(* IEC 61131-3 sources: Simulated-machine/integrations/openplc/thermal-plant-v4/pous/programs (part 2) *)

  (* Rising-edge plant trip matrix, matching examples/external_plc.py. *)
  IF turbine__discrete__tripped AND NOT i_turbine_trip_prev THEN
    generator__coil__breaker_open := TRUE;
    steam_valve__holding__manual_output := 0;
    generator__holding__primary_setpoint := 0;
  END_IF;
  i_turbine_trip_prev := turbine__discrete__tripped;
  IF boiler__discrete__tripped AND NOT i_boiler_trip_prev THEN
    boiler__holding__manual_output := 0;
    steam_valve__holding__manual_output := 0;
  END_IF;
  i_boiler_trip_prev := boiler__discrete__tripped;
  IF condenser__discrete__tripped AND NOT i_condenser_trip_prev THEN
    generator__holding__primary_setpoint := 0;
  END_IF;
  i_condenser_trip_prev := condenser__discrete__tripped;
  IF feedwater_pump__discrete__tripped AND NOT i_feedwater_pump_trip_prev THEN
    boiler__holding__manual_output := 0;
  END_IF;
  i_feedwater_pump_trip_prev := feedwater_pump__discrete__tripped;
  IF condensate_pump__discrete__tripped AND NOT i_condensate_pump_trip_prev THEN
    feedwater_pump__holding__manual_output := 2000;
  END_IF;
  i_condensate_pump_trip_prev := condensate_pump__discrete__tripped;
  IF steam_valve__discrete__tripped AND NOT i_steam_valve_trip_prev THEN
    boiler__holding__manual_output := 0;
  END_IF;
  i_steam_valve_trip_prev := steam_valve__discrete__tripped;

  (* Overspeed always closes the main steam valve, regardless of HMI demand. *)
  IF (turbine__input__speed_rpm > 3150) OR turbine__discrete__tripped THEN
    steam_valve__holding__manual_output := 0;
  END_IF;
END_PROGRAM
